TYPE ST_AXIS_MOVE_PROFILE :
STRUCT
	Velo	: REAL := 0;// Velocity
	Acc		: REAL := 0;// Acceleration
	Dec		: REAL := 0;// Deceleration
	Jerk	: REAL := 0;// Jerk
END_STRUCT
END_TYPE

(* stored: Version 1.1.0.1, ProductVersion 3.1.4024.12
   DUT ST_AXIS_MOVE_PROFILE: Id {5c1efe64-4c57-42fb-9340-801ec384ef19} *)
